PROGRAM IHM
VAR
		
	SafetyPLCIn 	AT %I*:BYTE;
	SafetyPLCOut 	AT %Q*:BYTE;
	
	sUrlAddressCamera : STRING;

	writeData:FB_WritePersistentData;
	t1:TON;
	bSavePersistent: BOOL;
	
	timer_login	: TON;
	
	Timer_Blink_1hz_1	: TON;
	Timer_Blink_1hz_2	: TON;
	
	b_contador		: BOOL;
	int_contador_10		: INT;
	
	
	PassoBtLigarDesligar	: INT;
	PassoBtReset			: INT;
	PassoMaquina			: INT;
	
END_VAR

(*=====================		STATUS DA MÁQUINA		======================*)

//Máquina em Alarme
IF (Alarmes.AlarmeGrave
	)THEN	
	MaquinaAlarme := TRUE;
ELSE
	MaquinaAlarme := FALSE;
END_IF	

(*=====================		LÓGICA DOS BOTÕES		======================*)

(*=====================		LIGAR E DESLIGAR		======================*)

//Condição de Bloqueio da Máquina de Estados - Botões Ligar e Desligar
IF (Alarmes.AlarmeGrave
	//OR Alarmes.AlarmeMedio
	//OR Alarmes.AlarmeLeve
	OR MaquinaModoManual
	) THEN
	PassoBtLigarDesligar := 1000;
	IhmBt_Desligar := TRUE;
	IhmBt_Ligar := FALSE;
	Flag_CondicoesIniciais := TRUE;
END_IF

// Máquina de Estados - Botões Ligar e Desligar
CASE PassoBtLigarDesligar OF

	//Passo 0 - Inicialização
	0: PassoBtLigarDesligar := 10;
	
	//Passo 10 - Botão Ligar
	10: IF IhmBt_Ligar THEN
			MaquinaLigada := TRUE;
			PassoBtLigarDesligar := 20;
			IhmBt_Ligar := TRUE;
			IhmBt_Desligar := FALSE;
		ELSIF NOT IhmBt_Ligar THEN
			IhmBt_Desligar := TRUE;
		END_IF
	
	//Passo 20 - Botão Desligar
	20: IF IhmBt_Desligar THEN
			MaquinaLigada := FALSE;
			PassoBtLigarDesligar := 1000;
			IhmBt_Ligar := FALSE;
			IhmBt_Desligar := TRUE;
		ELSIF NOT IhmBt_Ligar THEN
			IhmBt_Ligar := TRUE;
		END_IF
	
	//Passo 1000 - Finalização
	1000: PassoBtLigarDesligar := 0;

END_CASE

(*==========================		RESET		==========================*)

IF (InSolicitaReset OR IhmBt_Reset) THEN
	Reset := TRUE;
ELSE
	Reset := FALSE;
END_IF

(*=====================		MODO MANUAL / AUTO		======================*)

IF IhmBt_ManualAuto THEN
	IhmBt_ManualAuto_Text := 'MANUAL';
	IhmBt_ManualAuto_Color := TRUE;
	MaquinaModoManual := TRUE;
	MaquinaModoAuto := FALSE;
ELSE
	IhmBt_ManualAuto_Text := 'AUTO';
	IhmBt_ManualAuto_Color := FALSE;
	MaquinaModoManual := FALSE;
	MaquinaModoAuto := TRUE;
END_IF

(*========================================================================*)


(*========================================================================*)

//				Hora do Sistema					\\
	FB_HoraAtual (START := TRUE, TIMESTR => tempo);
	FB_HoraAtual (START := FALSE);
	TempoAtual := SYSTEMTIME_TO_DT (tempo);

t1(IN:= NOT t1.Q, PT:=T#1M);	
writeData(
	NETID:='' , 
	PORT:=851 , 
	START:= t1.Q OR bSavePersistent, 
	TMOUT:= T#10S, 
	MODE:= , 
	BUSY=> , 
	ERR=> ,  
	ERRID=> );	
	
	UserGroupName 	:= WSTRING_TO_STRING (visuelems.CurrentUserGroupName);
	UserGroupId		:= (visuelems.CurrentUserGroupId);

IF UserGroupId = 1 THEN
	UserName := WSTRING_TO_STRING(VisuElems.CurrentUserName);
	timer_login (in := FALSE);
	
ELSIF UserGroupId = 0 THEN
	timer_login (in := TRUE, pt := T#1S);	
	IF timer_login.Q THEN
		UserName := '';
		b_editar_receita := FALSE;
	END_IF
END_IF

(*///////////////////////////////			BLINK 0.25 HZ		\\\\\\\\\\\\\\\\\\\\\\\\\\\\\\\\\\\\\\\
IF IhmBt_Ligar THEN
	Timer_Blink_1hz_1 (IN := TRUE, PT := T#2S);	
END_IF

IF Timer_Blink_1hz_1.Q THEN
	Blink_1hz := TRUE;
	Timer_Blink_1hz_2 (IN := TRUE, PT := T#2S);
	IF Timer_Blink_1hz_2.Q THEN
		Blink_1hz := FALSE;
		Timer_Blink_1hz_1 (IN := FALSE);
		Timer_Blink_1hz_2 (IN := FALSE);
	END_IF
END_IF

	I2 := Blink_1hz;
	
	IF NOT b_contador AND Blink_1hz THEN
		b_contador := TRUE;
		Contador_Total := Contador_Total + 1;
		Contador_Pecas_Boas := Contador_Pecas_Boas + 1;
		int_contador_10 := int_contador_10 + 1;
	END_IF
	IF NOT Blink_1hz THEN
		b_contador := FALSE;
	END_IF
	
	IF int_contador_10 = 10 THEN
		int_contador_10 := 0;
		Contador_Pecas_Boas := Contador_Pecas_Boas - 1;
		Contador_Refugo := Contador_Refugo + 1;
	END_IF
*)	
	IF BT_ihm_zerar_contador THEN
		BT_ihm_zerar_contador := FALSE;
		Contador_Total := 0;
		Contador_PecasAprovadas := 0;
		Contador_PecasReprovadas := 0;
	END_IF

END_PROGRAM

(* stored: Version 1.1.0.1, ProductVersion 3.1.4024.11
   POU IHM: Id {c023c45d-cd98-427a-aae9-5d18b9d7be91}, SpecialFunc None *)
